FUNCTION_BLOCK FB_RemoteInterface
VAR_INPUT
	txUdp : ST_TxUdpRemote;
END_VAR
VAR_OUTPUT
	recvCounter : DINT := 0;
END_VAR
VAR
	// Udp connection
	{attribute 'tc_no_symbol'}
	udpClient : FB_UdpClient('', 0, 0, 0, 0, 0, 0);	// Dummy constructor
END_VAR

// Update Udp client
udpClient();

METHOD FB_exit : BOOL
VAR_INPUT
	bInCopyCode : BOOL; // if TRUE, the exit method is called for exiting an instance that is copied afterwards (online change).
END_VAR
END_METHOD

METHOD FB_init : BOOL
VAR_INPUT
	bInitRetains : BOOL; // if TRUE, the retain variables are initialized (warm start / cold start)
	bInCopyCode : BOOL;  // if TRUE, the instance afterwards gets moved into the copy code (online change)
	
	// Init variables
	_remoteIpAddr : T_Ipv4Addr;
	_remotePort : UINT;
	_localPort : UINT;
END_VAR
// Initilize udpClient
udpClient.FB_init(
	bInitRetains,
	bInCopyCode,
	_remoteIpAddr,
	_remotePort,
	_localPort,
	SIZEOF(recvCounter),
	ADR(recvCounter),
	SIZEOF(txUdp),
	ADR(txUdp)
);
END_METHOD

METHOD FB_reinit : BOOL
VAR_INPUT
END_VAR
END_METHOD

END_FUNCTION_BLOCK

(* stored: Version 1.1.0.1, ProductVersion 3.1.4022.7
   POU FB_RemoteInterface: Id {876c2b91-df3c-4683-9fd3-7a3048a99a09}, SpecialFunc None
   Method FB_exit: Id {8f02c622-0e73-4bd7-94f0-589e37e92221}
   Method FB_init: Id {6ef0140a-757a-433f-b860-bfc093351cf9}
   Method FB_reinit: Id {4fd06a20-81e1-4ab4-9bba-7c79e2cd39ec} *)
